FUNCTION_BLOCK AnalogDevice_1 IMPLEMENTS I_AnalogDevice
VAR
	Q AT%I* : INT;
	rampUp		: RampUp;
	rampDown	: RampDown;
	_value		: REAL;
	_zeroIn		: REAL;
	_zeroOut    : REAL;
	_spanIn     : REAL;
	_spanOut    : REAL;
	_PLC_CYCLE_TIME_ms	: REAL;
	
END_VAR


	Q	:=	REAL_TO_INT(_value);

METHOD DecreaseValue
VAR_INPUT
	EN			: BOOL;
	RampDownTime: TIME;
END_VAR

	rampDown(
		IN					:= EN, 
		RampDownTime		:= RampDownTime, 
		Ramp_lowerLimit		:= _spanIn, 
		Ramp_upperLimit		:= _spanOut, 
		PLC_CYCLE_TIME_ms	:= _PLC_CYCLE_TIME_ms,
		output				:= _value, 
		InProgress			=> );
END_METHOD

METHOD FB_init : BOOL
VAR_INPUT
	bInitRetains : BOOL; // if TRUE, the retain variables are initialized (warm start / cold start)
	bInCopyCode : BOOL;  // if TRUE, the instance afterwards gets moved into the copy code (online change)
	ZeroIn		: REAL;
	ZeroOut    : REAL;
	SpanIn     : REAL;
	SpanOut    : REAL;	
	PLC_CYCLE_TIME_ms: REAL;
END_VAR

	_zeroIn		:=	ZeroIn;
	_zeroOut    :=	ZeroOut;
	_spanIn     :=	SpanIn;
	_spanOut    :=	SpanOut;
	_PLC_CYCLE_TIME_ms	:=	PLC_CYCLE_TIME_ms;
END_METHOD

METHOD IncreaseValue
VAR_INPUT
	EN			: BOOL;
	RampUpTime: TIME;
END_VAR

	rampUp(
		IN					:= EN, 
		RampUpTime			:= RampUpTime, 
		Ramp_lowerLimit		:= _spanIn, 
		Ramp_upperLimit		:= _spanOut, 
		PLC_CYCLE_TIME_ms	:= _PLC_CYCLE_TIME_ms,
		output				:= _value, 
		InProgress			=> );
END_METHOD

METHOD Off
VAR_INPUT
END_VAR

	_value	:=	_spanIn;
END_METHOD

METHOD On
VAR_INPUT
END_VAR

	_value	:=	_spanOut;
END_METHOD

METHOD SetValue
VAR_INPUT
	value: INT;

END_VAR

	_value	:=	F_Scaling(Variable_In:= value, Input_min:= _zeroIn, Input_max:= _zeroOut, Output_min:= _spanIn, Output_max:= _spanOut);
END_METHOD

PROPERTY Status : INT
GET

	Status	:=	REAL_TO_INT(F_Scaling(Variable_In:= _value, Input_min:= _spanIn, Input_max:= _spanOut, Output_min:= _zeroIn, Output_max:= _zeroOut));
END_GET
END_PROPERTY

END_FUNCTION_BLOCK

(* stored: Version 1.1.0.1, ProductVersion 3.1.4024.13
   POU AnalogDevice_1: Id {f09fcb2f-4f22-428b-b43e-d378def66a76}, SpecialFunc None
   Method DecreaseValue: Id {1dbe2645-27ca-4c0b-9913-3367073bc373}
   Method FB_init: Id {93bbc8b2-1671-4e1e-bd3b-a3578e6691de}
   Method IncreaseValue: Id {07c1ec4d-4dc6-4d4a-ae5f-a753f98591cf}
   Method Off: Id {60c0fb48-4a5b-4323-a58f-9cd5d8cf58ef}
   Method On: Id {199d83c9-6a28-4821-89df-1797a1e473cc}
   Method SetValue: Id {7dd60c78-5fa1-4489-8fe2-7fea3222996c}
   Property Status: Id {28cf181b-e01b-458e-968c-506cd9acad39}
   Get Get: Id {62c18809-148b-4796-badd-d3f296644378} *)
